(* PLC project Unnamed, Unknown Unnamed 1 *)
(* stored: creationDateTime 2022-11-02T12:49:46, modificationDateTime 2022-11-15T16:38:04 *)

PROGRAM tcp_socket
  VAR
    TCP_Connect0 : TCP_CONNECT;
    connected : BOOL;
    socket_id : INT;
    pulse : BOOL;
    TON0 : TON;
    TOF0 : TOF;
    TCP_Send0 : TCP_SEND;
    TCP_Receive0 : TCP_RECEIVE;
    Received_bytes : INT;
    Received_msg : STRING;
    send_hi_back : BOOL;
    TCP_Send1 : TCP_SEND;
  END_VAR
  VAR  (* added by the conversion: wires and edge detectors of the diagram *)
    R_TRIG1 : R_TRIG;
    R_TRIG2 : R_TRIG;
  END_VAR

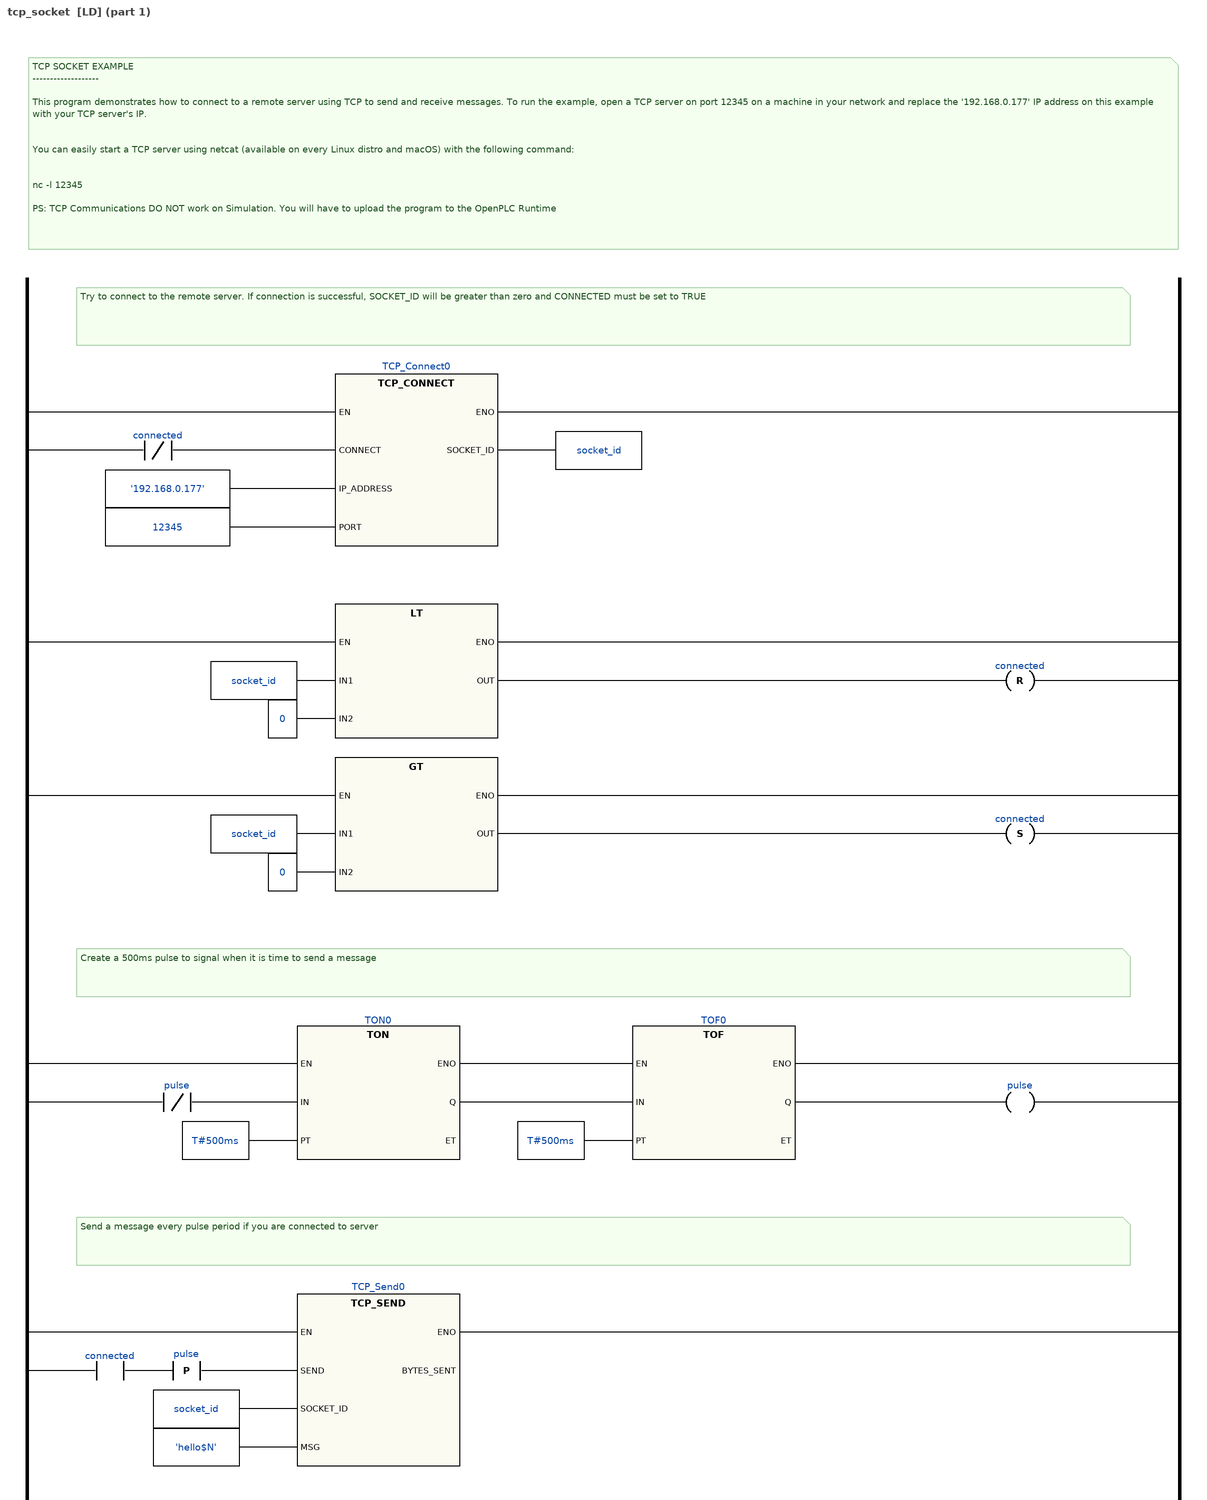
(* LD diagram, written out as Structured Text *)
(* TCP SOCKET EXAMPLE
-------------------

This program demonstrates how to connect to a remote server using TCP to send and receive messages. To run the example, open a TCP server on port 12345 on a machine in your network and replace the '192.168.0.177' IP address on this example with your TCP server's IP.


You can easily start a TCP server using netcat (available on every Linux distro and macOS) with the following command:


nc -l 12345

PS: TCP Communications DO NOT work on Simulation. You will have to upload the program to the OpenPLC Runtime *)
(* Try to connect to the remote server. If connection is successful, SOCKET_ID will be greater than zero and CONNECTED must be set to TRUE *)
TCP_Connect0(CONNECT := NOT connected, IP_ADDRESS := '192.168.0.177', PORT := 12345);
socket_id := TCP_Connect0.SOCKET_ID;
IF socket_id < 0 THEN connected := FALSE; END_IF;
IF socket_id > 0 THEN connected := TRUE; END_IF;
(* Create a 500ms pulse to signal when it is time to send a message *)
TON0(IN := NOT pulse, PT := T#500ms);
TOF0(EN := TON0.ENO, IN := TON0.Q, PT := T#500ms);
pulse := TOF0.Q;
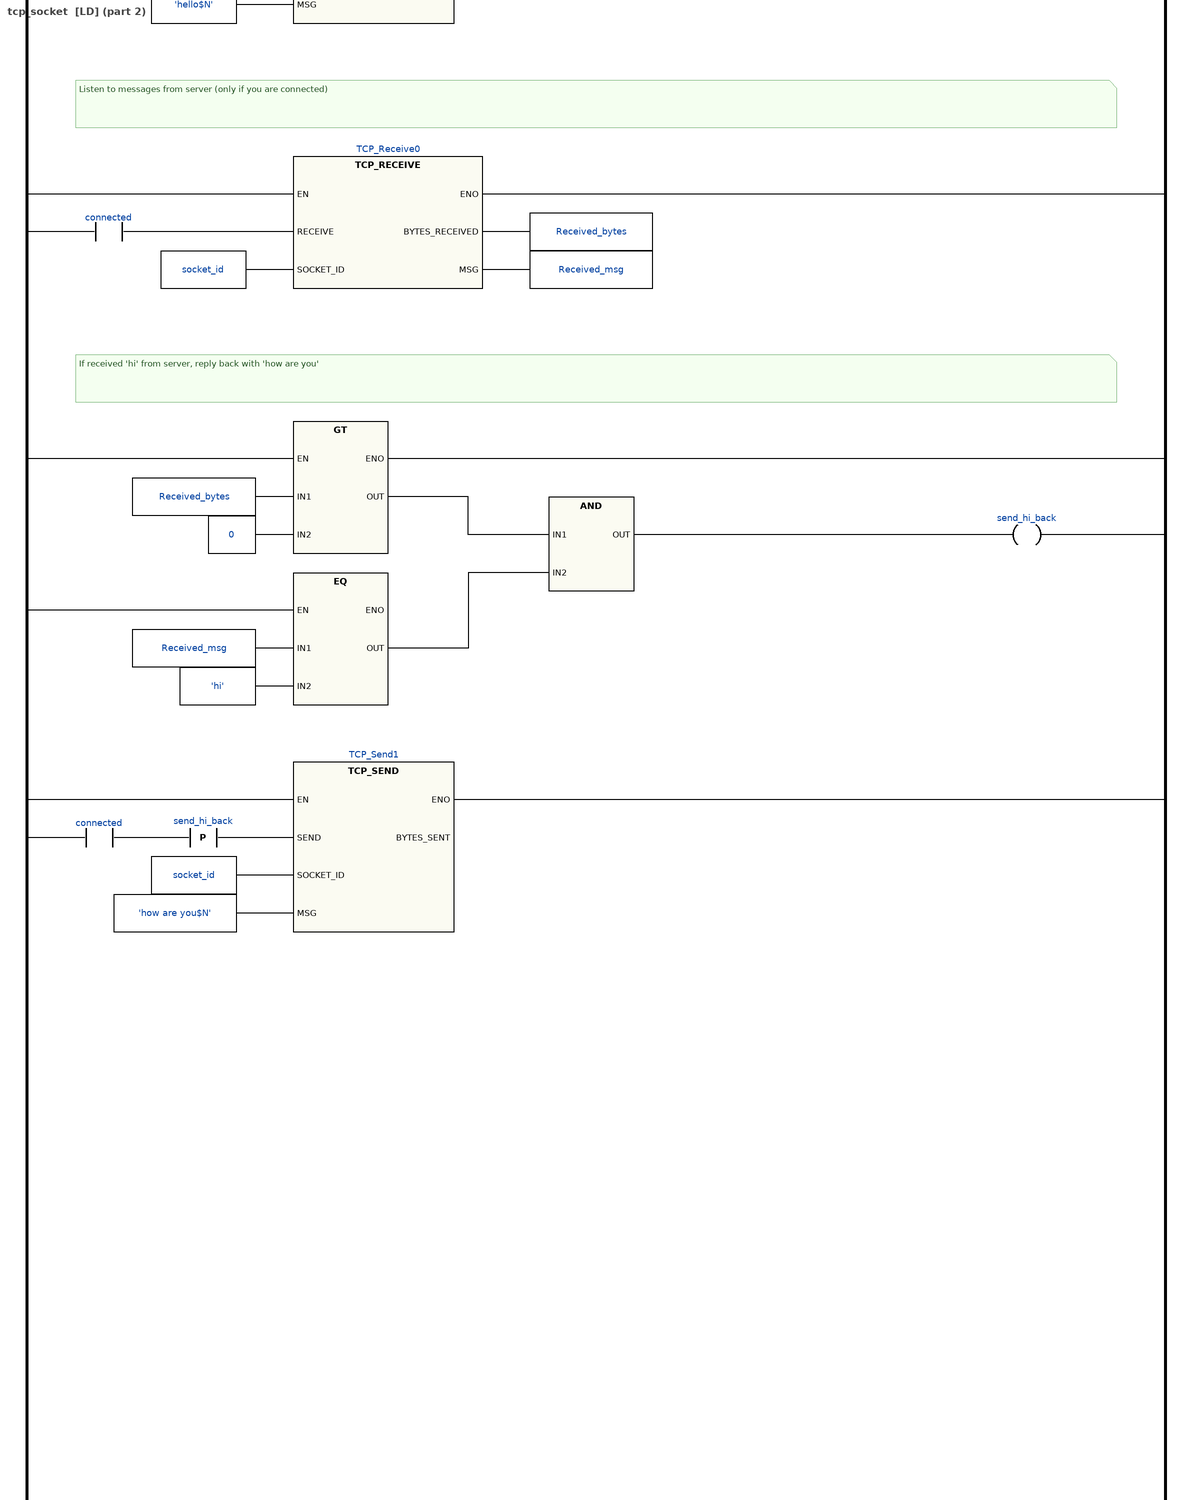
(* Send a message every pulse period if you are connected to server *)
(* Listen to messages from server (only if you are connected) *)
TCP_Receive0(RECEIVE := connected, SOCKET_ID := socket_id);
Received_bytes := TCP_Receive0.BYTES_RECEIVED;
Received_msg := TCP_Receive0.MSG;
(* If received 'hi' from server, reply back with 'how are you' *)
send_hi_back := Received_bytes > 0 AND Received_msg = 'hi';
R_TRIG1(CLK := pulse);
TCP_Send0(SEND := connected AND R_TRIG1.Q, SOCKET_ID := socket_id, MSG := 'hello$N');
R_TRIG2(CLK := send_hi_back);
TCP_Send1(SEND := connected AND R_TRIG2.Q, SOCKET_ID := socket_id, MSG := 'how are you$N');
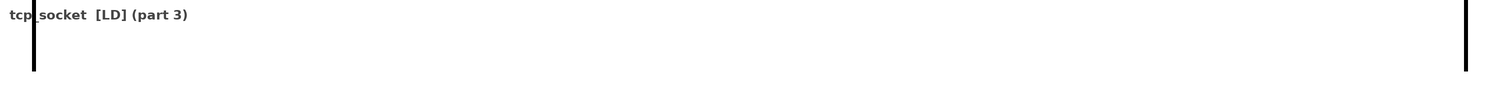
END_PROGRAM

CONFIGURATION Config0
  RESOURCE Res0 ON PLC
    TASK task0(INTERVAL := T#20ms, PRIORITY := 0);
    PROGRAM instance0 WITH task0 : tcp_socket;
  END_RESOURCE
END_CONFIGURATION
